// Mitsubishi GX Works2 project: 順次回路1   PLC: Q03UDV

PROGRAM MAIN
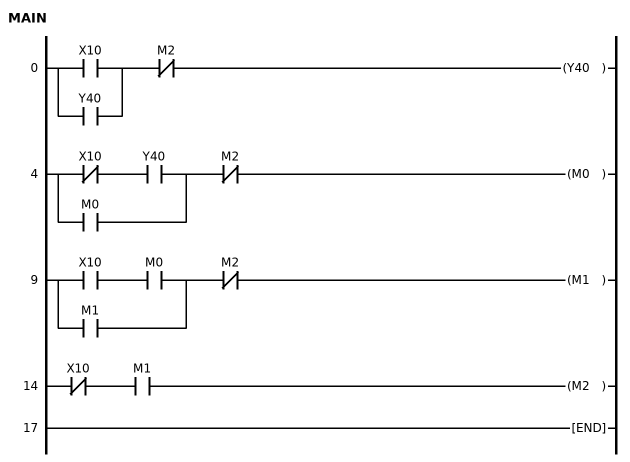
0     LD      X10
      OR      Y40
      ANI     M2
      OUT     Y40
4     LDI     X10
      AND     Y40
      OR      M0
      ANI     M2
      OUT     M0
9     LD      X10
      AND     M0
      OR      M1
      ANI     M2
      OUT     M1
14    LDI     X10
      AND     M1
      OUT     M2
17    END
END_PROGRAM
